// Mitsubishi GX Works2 project: hung_creat_plc_dich_bit_ver5   PLC: FX3U/FX3UC

PROGRAM MAIN
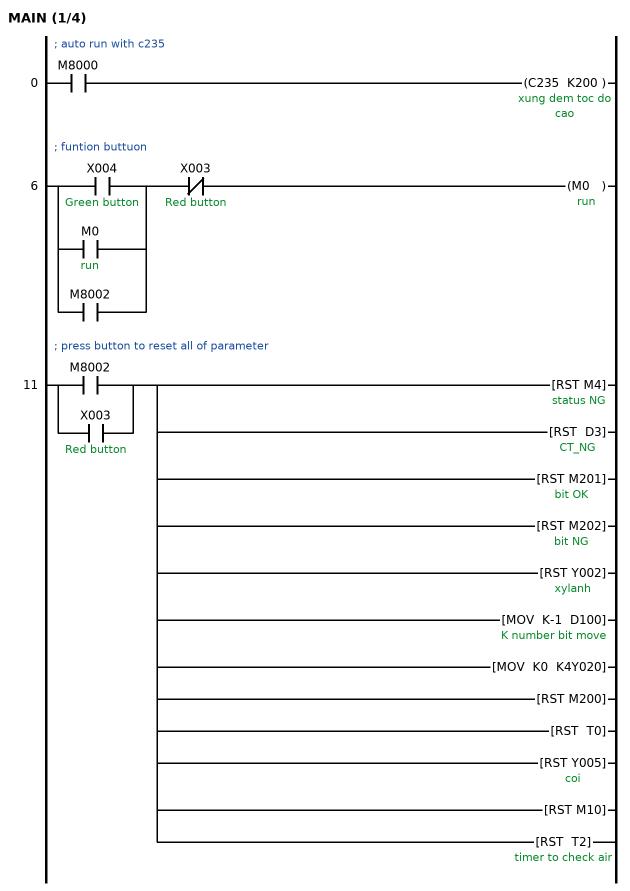
; auto run with c235
0     LD      M8000
      OUT     C235 K200  ; xung dem toc do  cao
; funtion buttuon
6     LD      X004  ; Green button
      OR      M0  ; run
      OR      M8002
      ANI     X003  ; Red button
      OUT     M0  ; run
; press button to reset all of parameter
11    LD      M8002
      OR      X003  ; Red button
      RST     M4  ; status NG
      RST     D3  ; CT_NG
      RST     M201  ; bit OK
      RST     M202  ; bit NG
      RST     Y002  ; xylanh
      MOV     K-1 D100  ; K number bit move
      MOV     K0 K4Y020  ; move right
      RST     M200
      RST     T0
      RST     Y005  ; coi
      RST     M10
      RST     T2  ; timer to check air
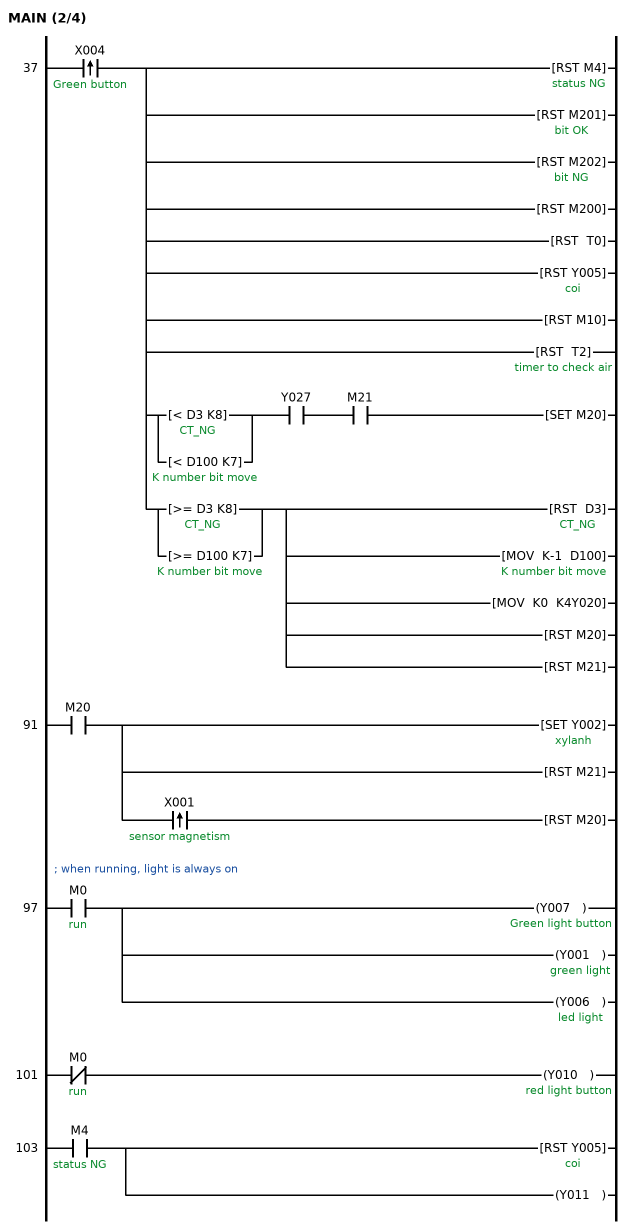
37    LDP     X004  ; Green button
      RST     M4  ; status NG
      RST     M201  ; bit OK
      RST     M202  ; bit NG
      RST     M200
      RST     T0
      RST     Y005  ; coi
      RST     M10
      RST     T2  ; timer to check air
      MPS
      LD<     D3 K8  ; CT_NG
      OR<     D100 K7  ; K number bit move
      ANB
      AND     Y027
      AND     M21
      SET     M20
      MPP
      LD>=    D3 K8  ; CT_NG
      OR>=    D100 K7  ; K number bit move
      ANB
      RST     D3  ; CT_NG
      MOV     K-1 D100
      MOV     K0 K4Y020
      RST     M20
      RST     M21
91    LD      M20
      SET     Y002  ; xylanh
      RST     M21
      ANDP    X001  ; sensor magnetism
      RST     M20
; when running, light is always on
97    LD      M0  ; run
      OUT     Y007  ; Green light button
      OUT     Y001  ; green light
      OUT     Y006  ; led light
101   LDI     M0  ; run
      OUT     Y010  ; red light button
103   LD      M4  ; status NG
      RST     Y005  ; coi
      OUT     Y011
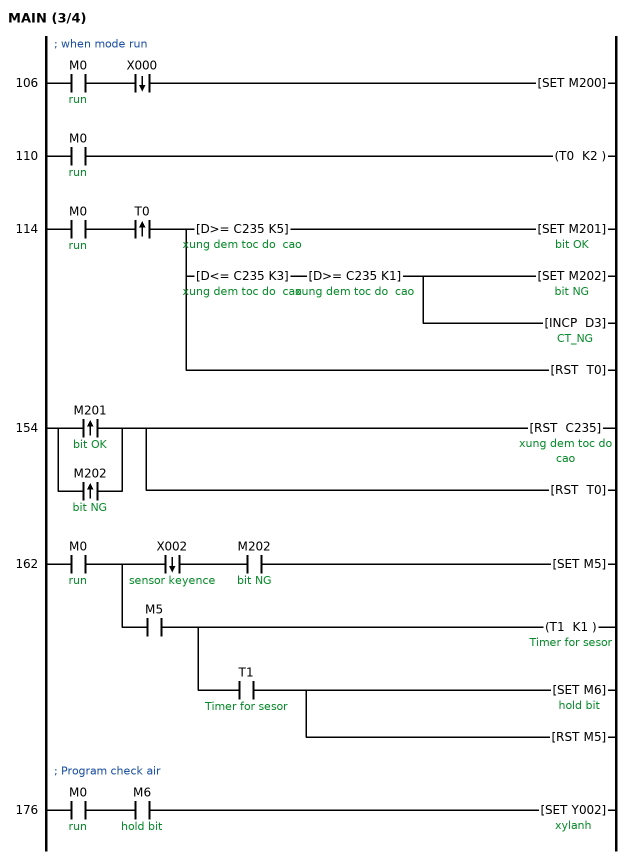
; when mode run
106   LD      M0  ; run
      ANDF    X000
      SET     M200
110   LD      M0  ; run
      OUT     T0 K2
114   LD      M0  ; run
      ANDP    T0
      MPS
      ANDD>=  C235 K5  ; xung dem toc do  cao
      SET     M201  ; bit OK
      MRD
      ANDD<=  C235 K3  ; xung dem toc do  cao
      ANDD>=  C235 K1  ; xung dem toc do  cao
      SET     M202  ; bit NG
      INCP    D3
      MPP
      RST     T0
154   LDP     M201  ; bit OK
      ORP     M202  ; bit NG
      RST     C235  ; xung dem toc do  cao
      RST     T0
162   LD      M0  ; run
      MPS
      ANDF    X002  ; sensor keyence
      AND     M202  ; bit NG
      SET     M5
      MPP
      AND     M5
      OUT     T1 K1  ; Timer for sesor
      AND     T1  ; Timer for sesor
      SET     M6  ; hold bit
      RST     M5
; Program check air
176   LD      M0  ; run
      AND     M6  ; hold bit
      SET     Y002  ; xylanh
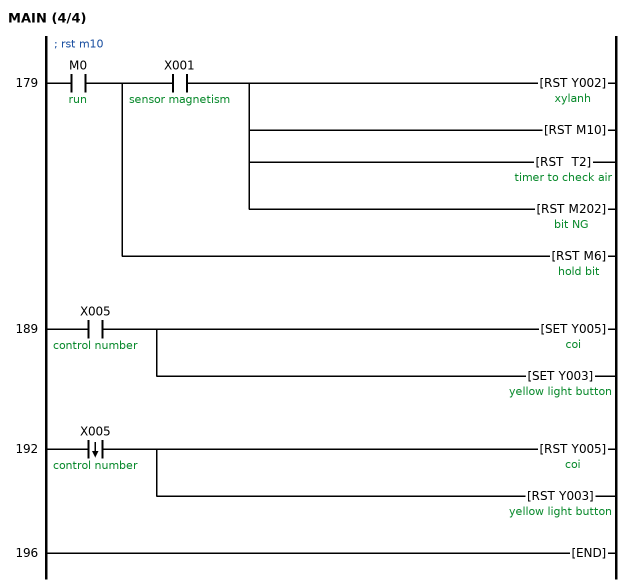
; rst m10
179   LD      M0  ; run
      MPS
      AND     X001  ; sensor magnetism
      RST     Y002  ; xylanh
      RST     M10
      RST     T2  ; timer to check air
      RST     M202  ; bit NG
      MPP
      RST     M6  ; hold bit
189   LD      X005  ; control number
      SET     Y005  ; coi
      SET     Y003  ; yellow light button
192   LDF     X005  ; control number
      RST     Y005  ; coi
      RST     Y003  ; yellow light button
196   END
END_PROGRAM

// device comments not shown above
D0  ; CT
Y000  ; red light
M3  ; bit reset NG and OK
M100  ; BIT TO MOVE
M300  ; timer for left bit
